TYPE (* Event type of the Arrowhead Framework *)
  (* Standard: 61499-2; Description: Copyright (c) 2019 fortiss GmbH This program and the accompanying materials are made available under the terms of the Eclipse Public License 2.0 which is available at https://www.eclipse.org/legal/epl-2.0/ SPDX-License-Identifier: EPL-2.0 *)
  (* Version 1.0, 2019-09-17, Jose Cabral, fortiss GmbH *)
  (* ASN.1 tag APPLICATION 1 *)
  ArrowheadEvent : STRUCT
    type : WSTRING; (* The type of the event, an event ID of sorts. *)
    payload : WSTRING; (* String data of the event. *)
    timestamp : DATE_AND_TIME; (* Date and time of the event. *)
    eventMetadata : ARRAY [0..9] OF WSTRING; (* Key=value pairs of additional data about the event. *)
  END_STRUCT;
END_TYPE
